// TwinCAT 3 PLC project RecipeServer_v2
// ProgramVersion: 3.1.4023.0
// libraries:
//   StringUtils, * (System)
//   Tc2_Standard, * (Beckhoff Automation GmbH)
//   Tc2_System, * (Beckhoff Automation GmbH)
//   Tc2_Utilities, * (Beckhoff Automation GmbH)
//   Tc3_Database, * (Beckhoff Automation GmbH)
//   Tc3_EventLogger, * (Beckhoff Automation GmbH)
//   Tc3_Module, * (Beckhoff Automation GmbH)
// project tree:
//   DUTs/Enumerations/ AllMaterialsEnum.TcTLEO
//   DUTs/ PaperInterval.TcDUT, PositionMaterials.TcDUT, PositionRotations.TcDUT, STRING_5K.TcDUT
//   GVLs/ BundleData.TcGVL, ExtrusionData.TcGVL, StrapWrapRecipe.TcGVL
//   GVLs/Constants/ GVL.TcGVL
//   / PlcTask.TcTTO
//   POUs/ AddRecipeToDatabase.TcPOU, MAIN.TcPOU, Validation.TcPOU
//   POUs/Functions/ ArrayFunctions.TcPOU, ConcatStrings.TcPOU
// (motion and I/O tree: see PLC project newplc)
// real-time tasks:
//   TASK PlcTask: cycle T#10ms, priority 20, ADS port 350
//   TASK PlcTask1: cycle T#10ms, priority 21, ADS port 351
//   TASK PlcTask2: cycle T#10ms, priority 22, ADS port 352
//   TASK PlcTask3: cycle T#10ms, priority 23, ADS port 353
//   TASK PlcTask4: cycle T#10ms, priority 24, ADS port 354
//   TASK PlcTask5: cycle T#10ms, priority 25, ADS port 355

CONFIGURATION RecipeServer_v2
    RESOURCE PLC ON TwinCAT3
        TASK PlcTask(INTERVAL := T#10ms, PRIORITY := 25);
        PROGRAM MAIN WITH PlcTask : MAIN;
    END_RESOURCE
END_CONFIGURATION

// ---- DUTs/Enumerations/AllMaterialsEnum.TcTLEO
{attribute 'qualified_only'}
{attribute 'strict'}
{attribute 'to_string'}
TYPE AllMaterialsEnum :
(
	//SIDES
	TOP, SIDES, BOTTOM,

	//CARDBOARD
	CAR20S, CAR20M, CAR20L, CAR28S, CAR28M, CAR28L, //base (flat)
	CAR20SF, CAR20MF, CAR20LF, CAR28SF, CAR28MF, CAR28LF, //single folded (L shape) - F
	CAR20SD, CAR20MD, CAR20LD, CAR28SD, CAR28MD, CAR28LD, //double folded (C shape) - D
	
	//CHIPBOARD
	CIP18, CIP54,
	
	//CORNER GUARD
	COR48,
	
	//PAPER
	PAP28,
	
	//WOOD BUNK
	WDT20, WDT22, WDT28, //top
	WDB20, WDB22, WDB28, //bottom
	WDS08, WDS10, WDS12, WDS14, WDS20, WDS22, WDS28, //side
	WDS8X8, WDS8X10, WDS12X12, WDS12X14, WDS20X10, WDS20X12, //side combined - X
	WDW20, WDW22, //special top (wide)
	
	size //number of materials
);
END_TYPE

// ---- DUTs/PaperInterval.TcDUT
TYPE PaperInterval :
STRUCT
	start : INT;
	end : INT;
	
	wrap : BOOL;
END_STRUCT
END_TYPE

// ---- DUTs/PositionMaterials.TcDUT
TYPE PositionMaterials :
STRUCT
	position : INT := 0; //default value is set to predefined constant if bundle needs less than 32 position material pairs
	
	top : STRING;
	left : STRING;
	right : STRING;
	bottom : STRING;
	
	topLeft : STRING;
	topLeftFold : INT;
	
	topRight : STRING;
	topRightFold : INT;
	
	bottomLeft : STRING;
	bottomLeftFold : INT;
	
	bottomRight : STRING;
	bottomRightFold : INT;
	
	numWrapPoints : INT;
	numWrapRotations : INT;
	
END_STRUCT
END_TYPE

// ---- DUTs/PositionRotations.TcDUT
TYPE PositionRotations : 
STRUCT
	position : INT;
	rotations : INT;
END_STRUCT
END_TYPE

// ---- DUTs/STRING_5K.TcDUT
TYPE STRING_5K : STRING(5000); END_TYPE

// ---- GVLs/BundleData.TcGVL
{attribute 'qualified_only'}
VAR_GLOBAL
	id : STRING;
	weight : REAL;
	
	length : REAL;
	height : REAL;
	width : REAL;
	
	pieces : USINT;
	layers : USINT;
	piecesPerLayer : USINT;
	
	requiredProcessing : ARRAY[0..3] OF BOOL;
END_VAR
VAR_GLOBAL CONSTANT
	//for requiredProcessing array
	AUTO_RE : INT := 0;
	MANUAL_RE : INT := 1;
	AUTO_SS : INT := 2;
	MANUAL_SS : INT := 3;
END_VAR

// ---- GVLs/ExtrusionData.TcGVL
{attribute 'qualified_only'}
VAR_GLOBAL	
	extrusionWeight : REAL;
	
	extrusionHeight : REAL;
	extrusionWidth : REAL;
END_VAR

// ---- GVLs/Constants/GVL.TcGVL
{attribute 'qualified_only'}
{attribute 'global_init_slot' := '45000'}
VAR_GLOBAL CONSTANT //first to compile
	maxMessages : UINT := 64;
	maxMaterials : DINT := 16; //max index, 0-15 are used with 16 as buffer
	
	//by materials
	Paper : ARRAY[1..1] OF STRING := ['PAP28'];
	CornerGuard : ARRAY[1..2] OF STRING := ['COR48', 'COR96'];
	
	CardboardSurfaces : ARRAY[1..6] OF STRING := ['CAR20S', 'CAR20M', 'CAR20L', 'CAR28S', 'CAR28M', 'CAR28L'];
	CardboardCorners : ARRAY[1..6] OF STRING := ['CAR20SF', 'CAR20MF', 'CAR20LF', 'CAR28SF', 'CAR28MF', 'CAR28LF'];
	
	Chipboard : ARRAY[1..2] OF STRING := ['CIP18', 'CIP54'];
	
	WoodBunkTop : ARRAY[1..5] OF STRING := ['WDT20', 'WDT22', 'WDT28', 'WDW20', 'WDW22'];
	WoodBunkSides : ARRAY[1..13] OF STRING := [	'WDS08', 'WDS10', 'WDS12', 'WDS14', 'WDS20','WDS22', 'WDS28', 'WDS8x8', 'WDS8x10', 'WDS12x12', 'WDS12x14', 'WDS20x10', 'WDS20x12'];										
	WoodBunkBottom : ARRAY[1..3] OF STRING := [	'WDB20', 'WDB22', 'WDB28'];
END_VAR

// ---- GVLs/StrapWrapRecipe.TcGVL
{attribute 'qualified_only'}
VAR_GLOBAL	
	//v2 - entries are in the format of position-material separated by material type
	faceCardboard : ARRAY[0..1] OF BOOL;
	facePaper : ARRAY[0..1] OF BOOL;
	
	TopPaper : ARRAY[0..GVL.maxMaterials] OF PaperInterval;
	LeftPaper : ARRAY[0..GVL.maxMaterials] OF PaperInterval;
	RightPaper : ARRAY[0..GVL.maxMaterials] OF PaperInterval;
	BottomPaper : ARRAY[0..GVL.maxMaterials] OF PaperInterval;
	
	Cardboard : ARRAY[0..GVL.maxMaterials] OF PositionMaterials;
	CornerGuard : ARRAY[0..GVL.maxMaterials] OF PositionMaterials;
	
	Chipboard : ARRAY[0..GVL.maxMaterials] OF PositionMaterials;
	WoodBunk : ARRAY[0..GVL.maxMaterials] OF PositionMaterials;
	
	PaperWrap : ARRAY[0..GVL.maxMaterials] OF PositionRotations;
	CardboardWrap : ARRAY[0..GVL.maxMaterials] OF PositionRotations;
END_VAR

// ---- POUs/MAIN.TcPOU
PROGRAM MAIN
VAR	
	generateRecipe : BOOL;
	
	addRecipeToDB : AddRecipeToDatabase;
	validator : Validation;
	arrayHelpers : ArrayFunctions;
	
	resetAddRecipeToDatabase : AddRecipeToDatabase;
	resetValidation : Validation;
	resetArrayFunctions : ArrayFunctions;
	
	start : BOOL := TRUE;
END_VAR

validator(); //real time error/warning message generator

IF generateRecipe THEN
	addRecipeToDB();
	
	IF addRecipeToDB.finished THEN
		reset();
		//reset all variables
		generateRecipe := FALSE;
		RETURN;
	END_IF
END_IF

METHOD reset : BOOL
VAR_INPUT
END_VAR
//reset FBs
MEMCPY(ADR(addRecipeToDB), ADR(resetAddRecipeToDatabase), SIZEOF(AddRecipeToDatabase));
MEMCPY(ADR(validator), ADR(resetValidation), SIZEOF(Validation));
MEMCPY(ADR(arrayHelpers), ADR(resetArrayFunctions), SIZEOF(ArrayFunctions));

//reset fields
BundleData.id := '';
BundleData.weight := 0;
BundleData.length := 0;
BundleData.height := 0;
BundleData.width := 0;
BundleData.pieces := 0;
BundleData.layers := 0;
BundleData.piecesPerLayer := 0;
MEMSET(ADR(BundleData.requiredProcessing), 0, SIZEOF(BundleData.requiredProcessing));

ExtrusionData.extrusionWeight := 0;
ExtrusionData.extrusionHeight := 0;
ExtrusionData.extrusionWidth := 0;

MEMSET(ADR(StrapWrapRecipe.facePaper), 0, SIZEOF(StrapWrapRecipe.facePaper));
MEMSET(ADR(StrapWrapRecipe.faceCardboard), 0, SIZEOF(StrapWrapRecipe.faceCardboard));
MEMSET(ADR(StrapWrapRecipe.TopPaper), 0, SIZEOF(StrapWrapRecipe.TopPaper));
MEMSET(ADR(StrapWrapRecipe.LeftPaper), 0, SIZEOF(StrapWrapRecipe.LeftPaper));
MEMSET(ADR(StrapWrapRecipe.RightPaper), 0, SIZEOF(StrapWrapRecipe.RightPaper));
MEMSET(ADR(StrapWrapRecipe.BottomPaper), 0, SIZEOF(StrapWrapRecipe.BottomPaper));
MEMSET(ADR(StrapWrapRecipe.Cardboard), 0, SIZEOF(StrapWrapRecipe.Cardboard));
MEMSET(ADR(StrapWrapRecipe.CornerGuard), 0, SIZEOF(StrapWrapRecipe.CornerGuard));
MEMSET(ADR(StrapWrapRecipe.Chipboard), 0, SIZEOF(StrapWrapRecipe.Chipboard));
MEMSET(ADR(StrapWrapRecipe.WoodBunk), 0, SIZEOF(StrapWrapRecipe.WoodBunk));
END_METHOD

END_PROGRAM

// ---- POUs/AddRecipeToDatabase.TcPOU
FUNCTION_BLOCK AddRecipeToDatabase //IMPLEMENTS I_TcEventBase
VAR
	cmd : ARRAY[0..19] OF STRING_5K;
	query : STRING_5K;
	
	fbSQLCommand : FB_SQLCommandEvt(sNetID := '', tTimeout := T#5S);
	fbSQLDatabase : FB_SQLDatabaseEvt (sNetID := '', tTimeout := T#5S);
	fbSQLResult: FB_SQLResultEvt(sNetID:='', tTimeout:=T#5S);
	
	eventString : STRING_5K;
	
	step : (CONNECT, READY, EXECUTE, FINISH);
END_VAR
VAR_OUTPUT
	finished : BOOL;
END_VAR

CASE step OF
	CONNECT:
		IF fbSQLDatabase.Connect(1) THEN
			IF NOT fbSqlDatabase.bError THEN
				step := READY;
			END_IF
		END_IF
		
	READY:
		IF fbSQLDatabase.CreateCmd(ADR(fbSQLCommand)) THEN
			step := EXECUTE;
		END_IF
	
	EXECUTE:
		query := completeQuery();
		IF fbSQLCommand.Execute(ADR(query), SIZEOF(query)) THEN
			step := FINISH;
		END_IF
		
	FINISH:
		IF fbSQLDatabase.Disconnect() THEN
			finished := TRUE;
		END_IF
END_CASE

METHOD completeQuery : STRING_5K
VAR_INST
	reqProcess : ARRAY[0..3] OF STRING_5K;
	
	queryOpening : STRING_5K := 'INSERT INTO "Bundle Data - Prototype" (BundleID, Weight, Length, Height, Width, Pieces, Layers, PiecesPerLayer, ExtrusionWeight, ExtrusionHeight, ExtrusionWidth, RequiredProcesses, Paper_top, Paper_sides, Paper_bottom, Cardboard, CornerGuard, Chipboard, WoodBunk) VALUES (';;
	queryClosing : STRING_5K := ')';
END_VAR
reqProcess[0] := TO_STRING(BundleData.requiredProcessing[0]);
reqProcess[1] := TO_STRING(BundleData.requiredProcessing[1]);
reqProcess[2] := TO_STRING(BundleData.requiredProcessing[2]);
reqProcess[3] := TO_STRING(BundleData.requiredProcessing[3]);


cmd[0] := TO_STRING(BundleData.id);
CONCAT2(ADR('$''), ADR(cmd[0]), ADR(cmd[0]), SIZEOF(cmd[0]));
CONCAT2(ADR(cmd[0]), ADR('$''), ADR(cmd[0]), SIZEOF(cmd[0]));

cmd[1] := TO_STRING(BundleData.weight);
cmd[2] := TO_STRING(BundleData.length);
cmd[3] := TO_STRING(BundleData.height);
cmd[4] := TO_STRING(BundleData.width);
cmd[5] := TO_STRING(BundleData.pieces);
cmd[6] := TO_STRING(BundleData.layers);
cmd[7] := TO_STRING(BundleData.piecesPerLayer);

cmd[8] := TO_STRING(ExtrusionData.extrusionWeight);
cmd[9] := TO_STRING(ExtrusionData.extrusionHeight);
cmd[10] := TO_STRING(ExtrusionData.extrusionWidth);

cmd[11] := ConcatStrings(reqProcess, 'ARRAY[', ']', ',');
//strap wrap recipe
cmd[12] := paperQuery(StrapWrapRecipe.TopPaper); //Paper_top
cmd[13] := paperQuery(StrapWrapRecipe.LeftPaper); //Paper_sides
cmd[14] := paperQuery(StrapWrapRecipe.RightPaper); //Paper_sides
cmd[15] := paperQuery(StrapWrapRecipe.BottomPaper); //Paper_sides

cmd[16] := materialQuery(StrapWrapRecipe.Cardboard);
cmd[17] := materialQuery(StrapWrapRecipe.CornerGuard);
cmd[18] := materialQuery(StrapWrapRecipe.Chipboard);
cmd[19] := materialQuery(StrapWrapRecipe.WoodBunk);

completeQuery := ConcatStrings(cmd, queryOpening, queryClosing, ',');
END_METHOD

METHOD materialQuery : STRING_5K
VAR_IN_OUT
	materialArr : ARRAY[*] OF PositionMaterials;
END_VAR
VAR_INST
	tempQuery : STRING_5K;
	
	position : STRING;
	top : STRING;
	left : STRING;
	right : STRING;
	bottom : STRING;
	
	topLeft : STRING;
	topLeftFold : STRING;
	topRight : STRING;
	topRightFold : STRING;
	
	bottomLeft : STRING;
	bottomLeftFold : STRING;
	bottomRight : STRING;
	bottomRightFold : STRING;
	
	i : DINT;
END_VAR
tempQuery := 'ARRAY[';

FOR i:=LOWER_BOUND(materialArr, 1) TO UPPER_BOUND(materialArr, 1) BY 1 DO
	position := TO_STRING(materialArr[i].position);
	
	top := TO_STRING(materialArr[i].top);
	left := TO_STRING(materialArr[i].left);
	right := TO_STRING(materialArr[i].right);
	bottom := TO_STRING(materialArr[i].bottom);
	
	topLeft := TO_STRING(materialArr[i].topLeft);
	topRight := TO_STRING(materialArr[i].topRight);
	bottomLeft := TO_STRING(materialArr[i].bottomLeft);
	bottomRight := TO_STRING(materialArr[i].bottomRight);
	
	topLeftFold := TO_STRING(materialArr[i].topLeftFold);
	topRightFold := TO_STRING(materialArr[i].topRightFold);
	bottomLeftFold := TO_STRING(materialArr[i].bottomLeftFold);
	bottomRightFold := TO_STRING(materialArr[i].bottomRightFold);
	
	IF top = '' AND left = '' AND right = '' AND bottom = '' AND topLeft = '' AND topRight = '' AND bottomLeft = '' AND bottomRight = '' THEN
		CONTINUE;
	END_IF
	
	IF i > LOWER_BOUND(materialArr, 1) THEN
		CONCAT2(ADR(tempQuery), ADR(', '), ADR(tempQuery), SIZEOF(tempQuery));
	END_IF

	CONCAT2(ADR(tempQuery), ADR('('), ADR(tempQuery), SIZEOF(tempQuery));
	CONCAT2(ADR(tempQuery), ADR(position), ADR(tempQuery), SIZEOF(tempQuery));
	CONCAT2(ADR(tempQuery), ADR(',$''), ADR(tempQuery), SIZEOF(tempQuery));
	
	CONCAT2(ADR(tempQuery), ADR(top), ADR(tempQuery), SIZEOF(tempQuery));
	CONCAT2(ADR(tempQuery), ADR('$', $''), ADR(tempQuery), SIZEOF(tempQuery));
	CONCAT2(ADR(tempQuery), ADR(left), ADR(tempQuery), SIZEOF(tempQuery));
	CONCAT2(ADR(tempQuery), ADR('$', $''), ADR(tempQuery), SIZEOF(tempQuery));
	CONCAT2(ADR(tempQuery), ADR(right), ADR(tempQuery), SIZEOF(tempQuery));
	CONCAT2(ADR(tempQuery), ADR('$', $''), ADR(tempQuery), SIZEOF(tempQuery));
	CONCAT2(ADR(tempQuery), ADR(bottom), ADR(tempQuery), SIZEOF(tempQuery));
	CONCAT2(ADR(tempQuery), ADR('$', $''), ADR(tempQuery), SIZEOF(tempQuery));
	
	CONCAT2(ADR(tempQuery), ADR(topLeft), ADR(tempQuery), SIZEOF(tempQuery));
	CONCAT2(ADR(tempQuery), ADR('$', $''), ADR(tempQuery), SIZEOF(tempQuery));
	CONCAT2(ADR(tempQuery), ADR(topRight), ADR(tempQuery), SIZEOF(tempQuery));
	CONCAT2(ADR(tempQuery), ADR('$', $''), ADR(tempQuery), SIZEOF(tempQuery));
	CONCAT2(ADR(tempQuery), ADR(bottomLeft), ADR(tempQuery), SIZEOF(tempQuery));
	CONCAT2(ADR(tempQuery), ADR('$', $''), ADR(tempQuery), SIZEOF(tempQuery));
	CONCAT2(ADR(tempQuery), ADR(bottomRight), ADR(tempQuery), SIZEOF(tempQuery));
	CONCAT2(ADR(tempQuery), ADR('$', '), ADR(tempQuery), SIZEOF(tempQuery));
	
	CONCAT2(ADR(tempQuery), ADR(topLeftFold), ADR(tempQuery), SIZEOF(tempQuery));
	CONCAT2(ADR(tempQuery), ADR(', '), ADR(tempQuery), SIZEOF(tempQuery));
	CONCAT2(ADR(tempQuery), ADR(topRightFold), ADR(tempQuery), SIZEOF(tempQuery));
	CONCAT2(ADR(tempQuery), ADR(', '), ADR(tempQuery), SIZEOF(tempQuery));
	CONCAT2(ADR(tempQuery), ADR(bottomLeftFold), ADR(tempQuery), SIZEOF(tempQuery));
	CONCAT2(ADR(tempQuery), ADR(', '), ADR(tempQuery), SIZEOF(tempQuery));
	CONCAT2(ADR(tempQuery), ADR(bottomRightFold), ADR(tempQuery), SIZEOF(tempQuery));
	
	CONCAT2(ADR(tempQuery), ADR(')'), ADR(tempQuery), SIZEOF(tempQuery));
END_FOR
CONCAT2(ADR(tempQuery), ADR(']::"PositionMaterials"[]'), ADR(tempQuery), SIZEOF(tempQuery));

materialQuery := tempQuery;
END_METHOD

METHOD paperQuery : STRING_5K
VAR_IN_OUT
	paperArr : ARRAY[*] OF PaperInterval;
END_VAR
VAR_INST
	tempQuery : STRING_5K;
	i : DINT;
	start : STRING;
	end : STRING;
	wrap : STRING;
END_VAR
tempQuery := 'ARRAY[';

FOR i:=LOWER_BOUND(paperArr, 1) TO UPPER_BOUND(paperArr, 1) BY 1 DO
	start := TO_STRING(paperArr[i].start);
	end := TO_STRING(paperArr[i].end);
	wrap := TO_STRING(paperArr[i].wrap);
	
	IF start = '0' AND end = '0' AND wrap = 'FALSE' THEN
		CONTINUE;
	END_IF
	
	IF i > LOWER_BOUND(paperArr, 1) THEN
		CONCAT2(ADR(tempQuery), ADR(','), ADR(tempQuery), SIZEOF(tempQuery));
	END_IF

	CONCAT2(ADR(tempQuery), ADR('('), ADR(tempQuery), SIZEOF(tempQuery));
	CONCAT2(ADR(tempQuery), ADR(start), ADR(tempQuery), SIZEOF(tempQuery));
	CONCAT2(ADR(tempQuery), ADR(','), ADR(tempQuery), SIZEOF(tempQuery));
	CONCAT2(ADR(tempQuery), ADR(end), ADR(tempQuery), SIZEOF(tempQuery));
	CONCAT2(ADR(tempQuery), ADR(','), ADR(tempQuery), SIZEOF(tempQuery));
	CONCAT2(ADR(tempQuery), ADR(wrap), ADR(tempQuery), SIZEOF(tempQuery));
	CONCAT2(ADR(tempQuery), ADR(')'), ADR(tempQuery), SIZEOF(tempQuery));
END_FOR
CONCAT2(ADR(tempQuery), ADR(']::"PaperInterval"[]'), ADR(tempQuery), SIZEOF(tempQuery));

paperQuery := tempQuery;
END_METHOD

END_FUNCTION_BLOCK

// ---- POUs/Functions/ConcatStrings.TcPOU
FUNCTION ConcatStrings : STRING_5K
VAR_IN_OUT
	stringsArr : ARRAY[*] OF STRING_5K;
END_VAR
VAR_INPUT
	opening : STRING_5K;
	closing : STRING_5K;
	separator : STRING_5K;
END_VAR
VAR
	fullString : STRING_5K;
	i : DINT := 0;	
END_VAR

fullString := opening; //opening segment

FOR i:=LOWER_BOUND(stringsArr, 1) TO UPPER_BOUND(stringsArr, 1)-1 BY 1 DO //first element to 2nd last element
	CONCAT2(ADR(fullString), ADR(stringsArr[i]), ADR(fullString), SIZEOF(fullString));
	CONCAT2(ADR(fullString), ADR(separator), ADR(fullString), SIZEOF(fullString));
END_FOR
CONCAT2(ADR(fullString), ADR(stringsArr[UPPER_BOUND(stringsArr, 1)]), ADR(fullString), SIZEOF(fullString)); //final element

CONCAT2(ADR(fullString), ADR(closing), ADR(fullString), SIZEOF(fullString)); //closing segment

concatStrings := fullString;

END_FUNCTION

// ---- POUs/Validation.TcPOU
FUNCTION_BLOCK Validation
VAR
	errors : ARRAY[0..GVL.maxMessages] OF STRING_5K;
	warnings : ARRAY[0..GVL.maxMessages] OF STRING_5K;

	tempErrors : ARRAY[0..GVL.maxMessages] OF STRING_5K;
	tempWarnings : ARRAY[0..GVL.maxMessages] OF STRING_5K;
	numErr : INT;
	numWarn : INT;
	
	bundleExists : BOOL;
		
	dbCheckStep : (CONNECT, READY, EXECUTE, FINISH);
	validationStep : (CHECK_EXISTING_BUNDLE, VALIDATE_DATA, FINISH_VALIDATION);
END_VAR

CASE validationStep OF
	CHECK_EXISTING_BUNDLE:
		IF checkExistingBundles() THEN
			validationStep := VALIDATE_DATA;
		END_IF
	
	VALIDATE_DATA:
		validateGeneralData(); //general data
		validateProcess(); //required processing
		validateMaterials(); //recipe
		
		validationStep := FINISH_VALIDATION;
		
	FINISH_VALIDATION: //copy temp to ADS and clear temp
		MEMCPY(ADR(errors), ADR(tempErrors), SIZEOF(errors));
		MEMCPY(ADR(warnings), ADR(tempWarnings), SIZEOF(warnings));
		
		MEMSET(ADR(tempErrors), 0, SIZEOF(tempErrors));
		MEMSET(ADR(tempWarnings), 0, SIZEOF(tempWarnings));
		numErr := 0;
		numWarn := 0;
		
		validationStep := CHECK_EXISTING_BUNDLE;
END_CASE

METHOD checkExistingBundles : BOOL
VAR_INST
	fbSQLCommand : FB_SQLCommandEvt(sNetID := '', tTimeout := T#5S);
	fbSQLDatabase : FB_SQLDatabaseEvt(sNetID := '', tTimeout := T#5S);
	fbSQLResult: FB_SQLResultEvt(sNetID := '', tTimeout := T#5S);
	
	
	cmd : ARRAY[0..2] OF STRING_5K;
	query : STRING_5K;
	tcMessage : I_TcMessage;
	existingID : STRING;
END_VAR
CASE dbCheckStep OF
	CONNECT:
		IF fbSQLDatabase.Connect(1) THEN
			IF NOT fbSqlDatabase.bError THEN
				dbCheckStep := READY;
			END_IF
		END_IF
		
	READY:
		IF fbSQLDatabase.CreateCmd(ADR(fbSQLCommand)) THEN
			dbCheckStep := EXECUTE;
		END_IF
	
	EXECUTE:
		cmd[0] := 'SELECT BundleID FROM "Bundle Data - Prototype" WHERE BundleID = $'';
		cmd[1] := TO_STRING(BundleData.id);
		cmd[2] := '$'';
		query := ConcatStrings(cmd, '', '', '');
		
		IF fbSQLCommand.ExecuteDataReturn(ADR(query), SIZEOF(query), ADR(fbSqlResult)) THEN
			dbCheckStep := FINISH;
		END_IF
		
	FINISH:
		fbSqlResult.Read(0, 1, ADR(existingID), SIZEOF(existingID), TRUE, FALSE);
		IF BundleData.id = existingID THEN
			bundleExists := TRUE;
		ELSE
			bundleExists := FALSE;
		END_IF
		IF fbSQLDatabase.Disconnect() THEN
			fbSqlResult.Release();
			checkExistingBundles := TRUE;
			dbCheckStep := CONNECT;
		END_IF
END_CASE
END_METHOD

{attribute 'TcRpcEnable'}
METHOD validateCardboard : BOOL
VAR_INST
	i : DINT;
END_VAR
FOR i:=0 TO GVL.maxMaterials BY 1 DO
	IF i > 0 THEN
		IF
			StrapWrapRecipe.Cardboard[i].position = StrapWrapRecipe.Cardboard[i-1].position 
			AND
			NOT(StrapWrapRecipe.Cardboard[i].position = 0 OR StrapWrapRecipe.Cardboard[i-1].position = 0)
		THEN
			tempWarnings[numWarn] := 'Cardboard: duplicate position';
			numWarn := numWarn + 1;
		END_IF
	END_IF
END_FOR
END_METHOD

{attribute 'TcRpcEnable'}
METHOD validateChipboard : BOOL
VAR_INST
	i : DINT;
END_VAR
FOR i:=0 TO GVL.maxMaterials BY 1 DO
	IF i > 0 THEN
		IF 
			StrapWrapRecipe.Chipboard[i].position = StrapWrapRecipe.Chipboard[i-1].position 
			AND
			NOT(StrapWrapRecipe.Chipboard[i].position = 0 OR StrapWrapRecipe.Chipboard[i-1].position = 0)
		THEN
			tempWarnings[numWarn] := 'Chipboard: duplicate position';
			numWarn := numWarn + 1;
		END_IF
	END_IF
END_FOR
END_METHOD

{attribute 'TcRpcEnable'}
METHOD validateCornerGuard : BOOL
VAR_INST
	i : DINT;
END_VAR
FOR i:=0 TO GVL.maxMaterials BY 1 DO
	IF i > 0 THEN
		IF 
			StrapWrapRecipe.CornerGuard[i].position = StrapWrapRecipe.CornerGuard[i-1].position 
			AND
			NOT(StrapWrapRecipe.CornerGuard[i].position = 0 OR StrapWrapRecipe.CornerGuard[i-1].position = 0)
		THEN
			tempWarnings[numWarn] := 'Corner Guard: duplicate position';
			numWarn := numWarn + 1;
		END_IF
	END_IF
END_FOR
END_METHOD

METHOD validateGeneralData : BOOL
IF BundleData.id = '' THEN //bundle id
	tempErrors[numErr] := 'ID missing';
	numErr := numErr + 1;
ELSIF BundleData.id <> '' AND bundleExists THEN
	tempWarnings[numWarn] := 'Bundle with entered ID already exists, proceeding will overwrite the existing recipe';
	numWarn := numWarn + 1;
END_IF

IF BundleData.weight = 0 THEN
	tempErrors[numErr] := 'Bundle weight missing';
	numErr := numErr + 1;
END_IF
IF BundleData.length = 0 OR BundleData.height = 0 OR BundleData.width = 0 THEN
	tempErrors[numErr] := 'Bundle dimension(s) missing';
	numErr := numErr + 1;
END_IF
IF BundleData.pieces = 0 OR BundleData.layers = 0 OR BundleData.piecesPerLayer = 0 THEN
	tempErrors[numErr] := 'Bundle layer dimension(s) missing';
	numErr := numErr + 1;
END_IF

IF Extrusiondata.extrusionWeight = 0 THEN
	tempErrors[numErr] := 'Extrusion weight missing';
	numErr := numErr + 1;
END_IF

IF Extrusiondata.extrusionHeight = 0 OR Extrusiondata.extrusionWidth = 0 THEN
	tempErrors[numErr] := 'Extrusion dimension(s) missing';
	numErr := numErr + 1;
END_IF
END_METHOD

{attribute 'TcRpcEnable'}
METHOD validateMaterials : BOOL
VAR_INST
	//fbSQLCommand : FB_SQLCommandEvt(sNetID := '', tTimeout := T#5S);
	//fbSQLDatabase : FB_SQLDatabaseEvt (sNetID := '', tTimeout := T#5S);
	//fbSQLResult: FB_SQLResultEvt(sNetID:='', tTimeout:=T#5S);
	
	
	
	
	//sqlResult : FB_SQLResult;
	
END_VAR

validatePaper();
validateCardboard();
validateCornerGuard();
validateChipboard();
validateWoodBunk();
END_METHOD

{attribute 'TcRpcEnable'}
METHOD validatePaper : BOOL
VAR_INST
	i : DINT;
END_VAR
FOR i:=0 TO GVL.maxMaterials BY 1 DO
	IF StrapWrapRecipe.TopPaper[i].start = 0 AND StrapWrapRecipe.TopPaper[i].end = 0 THEN //unused entry, do nothing and skip
		CONTINUE;
	END_IF
	
	IF StrapWrapRecipe.TopPaper[i].start >= StrapWrapRecipe.TopPaper[i].end THEN //invalid interval where start > end
		tempErrors[numErr] := 'Paper (Top): Start position must be less than end position';
		numErr := numErr + 1;
	END_IF
	
	IF i > 0 THEN
		IF StrapWrapRecipe.TopPaper[i].start < StrapWrapRecipe.TopPaper[i-1].end AND StrapWrapRecipe.TopPaper[i-1].end > 0 THEN //overlaps
			tempWarnings[numWarn] := 'Paper (Top): Overlapping segments';
			numWarn := numWarn + 1;
		ELSIF StrapWrapRecipe.TopPaper[i].start = StrapWrapRecipe.TopPaper[i-1].end AND StrapWrapRecipe.TopPaper[i-1].end > 0 THEN //adjacency
			tempWarnings[numWarn] := 'Paper (Top): Adjacent segments';
			numWarn := numWarn + 1;
		END_IF
	END_IF
END_FOR

FOR i:=0 TO GVL.maxMaterials BY 1 DO
	IF StrapWrapRecipe.LeftPaper[i].start = 0 AND StrapWrapRecipe.LeftPaper[i].end = 0 THEN //unused entry, do nothing and skip
		CONTINUE;
	END_IF
	
	IF StrapWrapRecipe.LeftPaper[i].start >= StrapWrapRecipe.LeftPaper[i].end THEN //invalid interval where start > end
		tempErrors[numErr] := 'Paper (Left): Start position must be less than end position';
		numErr := numErr + 1;
	END_IF
	
	IF i > 0 THEN
		IF StrapWrapRecipe.LeftPaper[i].start < StrapWrapRecipe.LeftPaper[i-1].end AND StrapWrapRecipe.LeftPaper[i-1].end > 0 THEN //overlaps
			tempWarnings[numWarn] := 'Paper (Left): Overlapping intervals, ignore if this is intended';
			numWarn := numWarn + 1;
		ELSIF StrapWrapRecipe.LeftPaper[i].start = StrapWrapRecipe.LeftPaper[i-1].end AND StrapWrapRecipe.LeftPaper[i-1].end > 0 THEN //adjacency
			tempWarnings[numWarn] := 'Paper (Left): Adjacent intervals can connected, ignore if this is intended';
			numWarn := numWarn + 1;
		END_IF
	END_IF
END_FOR

FOR i:=0 TO GVL.maxMaterials BY 1 DO
	IF StrapWrapRecipe.RightPaper[i].start = 0 AND StrapWrapRecipe.RightPaper[i].end = 0 THEN //unused entry, do nothing and skip
		CONTINUE;
	END_IF
	
	IF StrapWrapRecipe.RightPaper[i].start >= StrapWrapRecipe.RightPaper[i].end THEN //invalid interval where start > end
		tempErrors[numErr] := 'Paper (Right): Start position must be less than end position';
		numErr := numErr + 1;
	END_IF
	
	IF i > 0 THEN
		IF StrapWrapRecipe.RightPaper[i].start < StrapWrapRecipe.RightPaper[i-1].end AND StrapWrapRecipe.RightPaper[i-1].end > 0 THEN //overlaps
			tempWarnings[numWarn] := 'Paper (Right): Overlapping intervals, ignore if this is intended';
			numWarn := numWarn + 1;
		ELSIF StrapWrapRecipe.RightPaper[i].start = StrapWrapRecipe.RightPaper[i-1].end AND StrapWrapRecipe.RightPaper[i-1].end > 0 THEN //adjacency
			tempWarnings[numWarn] := 'Paper (Right): Adjacent intervals can connected, ignore if this is intended';
			numWarn := numWarn + 1;
		END_IF
	END_IF
END_FOR

FOR i:=0 TO GVL.maxMaterials BY 1 DO
	IF StrapWrapRecipe.BottomPaper[i].start = 0 AND StrapWrapRecipe.BottomPaper[i].end = 0 THEN //unused entry, do nothing and skip
		CONTINUE;
	END_IF
	
	IF StrapWrapRecipe.BottomPaper[i].start >= StrapWrapRecipe.BottomPaper[i].end THEN //invalid interval where start > end
		tempErrors[numErr] := 'Paper (Bottom): Start position must be less than end position';
		numErr := numErr + 1;
	END_IF
	
	IF i > 0 THEN
		IF StrapWrapRecipe.BottomPaper[i].start < StrapWrapRecipe.BottomPaper[i-1].end AND StrapWrapRecipe.BottomPaper[i-1].end > 0 THEN //overlaps
			tempWarnings[numWarn] := 'Paper (Bottom): Overlapping segments';
			numWarn := numWarn + 1;
		ELSIF StrapWrapRecipe.BottomPaper[i].start = StrapWrapRecipe.BottomPaper[i-1].end AND StrapWrapRecipe.BottomPaper[i-1].end > 0 THEN //adjacency
			tempWarnings[numWarn] := 'Paper (Bottom): Adjacent segments';
			numWarn := numWarn + 1;
		END_IF
	END_IF
END_FOR
END_METHOD

METHOD validateProcess : BOOL
VAR_INPUT
END_VAR
IF ( //if recipe exists but auto/manual strap and wrap is not selected
	StrapWrapRecipe.TopPaper[0].end > 0 OR 
	StrapWrapRecipe.LeftPaper[0].end > 0 OR 
	StrapWrapRecipe.RightPaper[0].end > 0 OR
	StrapWrapRecipe.BottomPaper[0].end > 0 OR 
	
	StrapWrapRecipe.Cardboard[0].top <> '' OR 
	StrapWrapRecipe.Cardboard[0].left <> '' OR 
	StrapWrapRecipe.Cardboard[0].right <> '' OR 
	StrapWrapRecipe.Cardboard[0].bottom <> '' OR 
	
	StrapWrapRecipe.Cardboard[0].topLeft <> '' OR 
	StrapWrapRecipe.Cardboard[0].topRight <> '' OR 
	StrapWrapRecipe.Cardboard[0].bottomLeft <> '' OR 
	StrapWrapRecipe.Cardboard[0].bottomRight <> '' OR 
	
	StrapWrapRecipe.CornerGuard[0].topLeft <> '' OR 
	StrapWrapRecipe.CornerGuard[0].topRight <> '' OR 
	StrapWrapRecipe.CornerGuard[0].bottomLeft <> '' OR 
	StrapWrapRecipe.CornerGuard[0].bottomRight <> '' OR 
	
	StrapWrapRecipe.Chipboard[0].top <> '' OR 
	StrapWrapRecipe.Chipboard[0].left <> '' OR 
	StrapWrapRecipe.Chipboard[0].right <> '' OR 
	StrapWrapRecipe.Chipboard[0].Bottom <> '' OR 

	StrapWrapRecipe.WoodBunk[0].top <> '' OR 
	StrapWrapRecipe.WoodBunk[0].left <> '' OR 
	StrapWrapRecipe.WoodBunk[0].right <> '' OR 
	StrapWrapRecipe.WoodBunk[0].Bottom <> '')
THEN
	IF NOT BundleData.requiredProcessing[BundleData.AUTO_SS] AND NOT BundleData.requiredProcessing[BundleData.MANUAL_SS] THEN
		tempErrors[numErr] := 'Recipe exists but strap and wrap processes are not selected (Auto/Manual Strap and Wrap)';
		numErr := numErr + 1;
	END_IF
ELSE //no recipe exists but auto/manual strap and wrap is selected
	IF BundleData.requiredProcessing[BundleData.AUTO_SS] OR BundleData.requiredProcessing[BundleData.MANUAL_SS] THEN
		tempWarnings[numWarn] := 'Strap and wrap processes are selected but there is no recipe, is this intended?';
		numWarn := numWarn + 1;
	END_IF
END_IF

	
IF //auto and manual strap/wrap are both selected
	(BundleData.requiredProcessing[BundleData.AUTO_RE] AND BundleData.requiredProcessing[BundleData.MANUAL_RE]) OR
	(BundleData.requiredProcessing[BundleData.AUTO_SS] AND BundleData.requiredProcessing[BundleData.MANUAL_SS])
THEN
	tempErrors[numErr] := 'Auto and Manual processes of the same type cannot be selected together';
	numErr := numErr + 1;
	
ELSIF //no processes selected
	NOT BundleData.requiredProcessing[BundleData.AUTO_RE] AND 
	NOT BundleData.requiredProcessing[BundleData.AUTO_SS] AND
	NOT BundleData.requiredProcessing[BundleData.MANUAL_RE] AND 
	NOT BundleData.requiredProcessing[BundleData.MANUAL_SS]
THEN
	tempWarnings[numWarn] := 'No processes are selected, is this intended?';
	numWarn := numWarn + 1;
END_IF
END_METHOD

{attribute 'TcRpcEnable'}
METHOD validateWoodBunk : BOOL
VAR_INST
	i : DINT;
END_VAR
FOR i:=0 TO GVL.maxMaterials BY 1 DO
	IF i > 0 THEN
		IF 
			StrapWrapRecipe.WoodBunk[i].position = StrapWrapRecipe.WoodBunk[i-1].position 
			AND
			NOT(StrapWrapRecipe.WoodBunk[i].position = 0 OR StrapWrapRecipe.WoodBunk[i-1].position = 0)
		THEN
			tempWarnings[numWarn] := 'Wood Bunk: duplicate position';
			numWarn := numWarn + 1;
		END_IF
	END_IF
END_FOR
END_METHOD

END_FUNCTION_BLOCK

// ---- POUs/Functions/ArrayFunctions.TcPOU
FUNCTION_BLOCK ArrayFunctions
VAR
	j : DINT;
END_VAR

{attribute 'TcRpcEnable'}
METHOD removeCardboard : BOOL
VAR_INPUT
	i : INT; //index to be removed
END_VAR
MEMMOVE(ADR(StrapWrapRecipe.Cardboard[i]), ADR(StrapWrapRecipe.Cardboard[i+1]), (GVL.maxMaterials-i)*SIZEOF(PositionMaterials));
StrapWrapRecipe.Cardboard[GVL.maxMaterials].position := 0;

StrapWrapRecipe.Cardboard[GVL.maxMaterials].top := '';
StrapWrapRecipe.Cardboard[GVL.maxMaterials].left := '';
StrapWrapRecipe.Cardboard[GVL.maxMaterials].right := '';
StrapWrapRecipe.Cardboard[GVL.maxMaterials].bottom := '';

StrapWrapRecipe.Cardboard[GVL.maxMaterials].topLeft := '';
StrapWrapRecipe.Cardboard[GVL.maxMaterials].topRight := '';
StrapWrapRecipe.Cardboard[GVL.maxMaterials].bottomLeft := '';
StrapWrapRecipe.Cardboard[GVL.maxMaterials].bottomRight := '';

StrapWrapRecipe.Cardboard[GVL.maxMaterials].topLeftFold := 0;
StrapWrapRecipe.Cardboard[GVL.maxMaterials].topRightFold := 0;
StrapWrapRecipe.Cardboard[GVL.maxMaterials].bottomLeftFold := 0;
StrapWrapRecipe.Cardboard[GVL.maxMaterials].bottomRightFold := 0;
END_METHOD

{attribute 'TcRpcEnable'}
METHOD removeChipboard : BOOL
VAR_INPUT
	i : INT; //index to be removed
END_VAR
MEMMOVE(ADR(StrapWrapRecipe.Chipboard[i]), ADR(StrapWrapRecipe.Chipboard[i+1]), (GVL.maxMaterials-i)*SIZEOF(PositionMaterials));
StrapWrapRecipe.Chipboard[GVL.maxMaterials].position := 0;

StrapWrapRecipe.Chipboard[GVL.maxMaterials].top := '';
StrapWrapRecipe.Chipboard[GVL.maxMaterials].left := '';
StrapWrapRecipe.Chipboard[GVL.maxMaterials].right := '';
StrapWrapRecipe.Chipboard[GVL.maxMaterials].bottom := '';

StrapWrapRecipe.Chipboard[GVL.maxMaterials].topLeft := '';
StrapWrapRecipe.Chipboard[GVL.maxMaterials].topRight := '';
StrapWrapRecipe.Chipboard[GVL.maxMaterials].bottomLeft := '';
StrapWrapRecipe.Chipboard[GVL.maxMaterials].bottomRight := '';

StrapWrapRecipe.Chipboard[GVL.maxMaterials].topLeftFold := 0;
StrapWrapRecipe.Chipboard[GVL.maxMaterials].topRightFold := 0;
StrapWrapRecipe.Chipboard[GVL.maxMaterials].bottomLeftFold := 0;
StrapWrapRecipe.Chipboard[GVL.maxMaterials].bottomRightFold := 0;
END_METHOD

{attribute 'TcRpcEnable'}
METHOD removeCornerGuard : BOOL
VAR_INPUT
	i : INT; //index to be removed
END_VAR
MEMMOVE(ADR(StrapWrapRecipe.CornerGuard[i]), ADR(StrapWrapRecipe.CornerGuard[i+1]), (GVL.maxMaterials-i)*SIZEOF(PositionMaterials));
StrapWrapRecipe.CornerGuard[GVL.maxMaterials].position := 0;

MEMSET(ADR(StrapWrapRecipe.CornerGuard[GVL.maxMaterials]), 0, SIZEOF(PositionMaterials));
END_METHOD

{attribute 'TcRpcEnable'}
METHOD removePaper: BOOL
VAR_INPUT
	face : STRING;
	i : DINT; //index to be removed
END_VAR
IF face = 'Top' THEN
	MEMMOVE(ADR(StrapWrapRecipe.TopPaper[i]), ADR(StrapWrapRecipe.TopPaper[i+1]), (GVL.maxMaterials-i)*SIZEOF(PaperInterval));
	StrapWrapRecipe.TopPaper[GVL.maxMaterials].start := 0;
	StrapWrapRecipe.TopPaper[GVL.maxMaterials].end := 0;
ELSIF face = 'Left' THEN
	MEMMOVE(ADR(StrapWrapRecipe.LeftPaper[i]), ADR(StrapWrapRecipe.LeftPaper[i+1]), (GVL.maxMaterials-i)*SIZEOF(PaperInterval));
	StrapWrapRecipe.LeftPaper[GVL.maxMaterials].start := 0;
	StrapWrapRecipe.LeftPaper[GVL.maxMaterials].end := 0;
ELSIF face = 'Right' THEN
	MEMMOVE(ADR(StrapWrapRecipe.RightPaper[i]), ADR(StrapWrapRecipe.RightPaper[i+1]), (GVL.maxMaterials-i)*SIZEOF(PaperInterval));
	StrapWrapRecipe.RightPaper[GVL.maxMaterials].start := 0;
	StrapWrapRecipe.RightPaper[GVL.maxMaterials].end := 0;
ELSIF face = 'Bottom' THEN
	MEMMOVE(ADR(StrapWrapRecipe.TopPaper[i]), ADR(StrapWrapRecipe.TopPaper[i+1]), (GVL.maxMaterials-i)*SIZEOF(PaperInterval));
	StrapWrapRecipe.BottomPaper[GVL.maxMaterials].start := 0;
	StrapWrapRecipe.BottomPaper[GVL.maxMaterials].end := 0;
END_IF
END_METHOD

{attribute 'TcRpcEnable'}
METHOD removeWoodBunk : BOOL
VAR_INPUT
	i : INT; //index to be removed
END_VAR
MEMMOVE(ADR(StrapWrapRecipe.WoodBunk[i]), ADR(StrapWrapRecipe.WoodBunk[i+1]), (GVL.maxMaterials-i)*SIZEOF(PositionMaterials));
StrapWrapRecipe.WoodBunk[GVL.maxMaterials].position := 0;

StrapWrapRecipe.WoodBunk[GVL.maxMaterials].top := '';
StrapWrapRecipe.WoodBunk[GVL.maxMaterials].left := '';
StrapWrapRecipe.WoodBunk[GVL.maxMaterials].right := '';
StrapWrapRecipe.WoodBunk[GVL.maxMaterials].bottom := '';

StrapWrapRecipe.WoodBunk[GVL.maxMaterials].topLeft := '';
StrapWrapRecipe.WoodBunk[GVL.maxMaterials].topRight := '';
StrapWrapRecipe.WoodBunk[GVL.maxMaterials].bottomLeft := '';
StrapWrapRecipe.WoodBunk[GVL.maxMaterials].bottomRight := '';

StrapWrapRecipe.WoodBunk[GVL.maxMaterials].topLeftFold := 0;
StrapWrapRecipe.WoodBunk[GVL.maxMaterials].topRightFold := 0;
StrapWrapRecipe.WoodBunk[GVL.maxMaterials].bottomLeftFold := 0;
StrapWrapRecipe.WoodBunk[GVL.maxMaterials].bottomRightFold := 0;
END_METHOD

{attribute 'TcRpcEnable'}
METHOD sortEntries : BOOL
sortPositionMaterials(StrapWrapRecipe.Cardboard);
sortPositionMaterials(StrapWrapRecipe.CornerGuard);
sortPositionMaterials(StrapWrapRecipe.Chipboard);
sortPositionMaterials(StrapWrapRecipe.WoodBunk);

sortPaperIntervals(StrapWrapRecipe.TopPaper);
sortPaperIntervals(StrapWrapRecipe.LeftPaper);
sortPaperIntervals(StrapWrapRecipe.RightPaper);
sortPaperIntervals(StrapWrapRecipe.BottomPaper);
END_METHOD

METHOD sortPaperIntervals : BOOL
VAR_IN_OUT
	arr : ARRAY[*] OF PaperInterval;
END_VAR
VAR_INST
	i : DINT;
	j : DINT;
	temp : PaperInterval;
END_VAR
FOR i:=LOWER_BOUND(arr, 1) TO UPPER_BOUND(arr, 1) BY 1 DO
	FOR j:=LOWER_BOUND(arr, 1) TO UPPER_BOUND(arr, 1)-i-1 BY 1 DO
		IF 
			(arr[j].start = 0 AND arr[j].end = 0) //unused entry
			OR 
			arr[j].start > arr[j+1].start AND //out of order and both entries are valid
			NOT(arr[j+1].start = 0 AND arr[j+1].end = 0)
		THEN //unused entry or out of order
			MEMCPY(ADR(temp), ADR(arr[j]), SIZEOF(PaperInterval));
			MEMCPY(ADR(arr[j]), ADR(arr[j+1]), SIZEOF(PaperInterval));
			MEMCPY(ADR(arr[j+1]), ADR(temp), SIZEOF(PaperInterval));
		END_IF
	END_FOR
END_FOR
END_METHOD

METHOD sortPositionMaterials : BOOL
VAR_IN_OUT
	arr : ARRAY[*] OF PositionMaterials;
END_VAR
VAR_INST
	i : DINT;
	j : DINT;
	temp : PositionMaterials;
END_VAR
FOR i:=LOWER_BOUND(arr, 1) TO UPPER_BOUND(arr, 1)-1 BY 1 DO
	FOR j:=LOWER_BOUND(arr, 1) TO UPPER_BOUND(arr, 1)-i-1 BY 1 DO
		IF //unused entry
			arr[j].top = '' AND arr[j].left = '' AND arr[j].right = '' AND arr[j].bottom = '' AND 
			arr[j].topRight = '' AND arr[j].topLeft = '' AND arr[j].bottomRight = '' AND arr[j].bottomLeft = ''
		THEN //unused entry
			arr[j].position := 0; //set position to 0
			MEMCPY(ADR(temp), ADR(arr[j]), SIZEOF(PositionMaterials));
			MEMCPY(ADR(arr[j]), ADR(arr[j+1]), SIZEOF(PositionMaterials));
			MEMCPY(ADR(arr[j+1]), ADR(temp), SIZEOF(PositionMaterials));
		ELSIF //out of order and both entries are valid
			arr[j].position > arr[j+1].position AND 
			NOT(
				arr[j+1].top = '' AND arr[j+1].left = '' AND arr[j+1].right = '' AND arr[j+1].bottom = '' AND 
				arr[j+1].topRight = '' AND arr[j+1].topLeft = '' AND arr[j+1].bottomRight = '' AND arr[j+1].bottomLeft = '')
		THEN
			MEMCPY(ADR(temp), ADR(arr[j]), SIZEOF(PositionMaterials));
			MEMCPY(ADR(arr[j]), ADR(arr[j+1]), SIZEOF(PositionMaterials));
			MEMCPY(ADR(arr[j+1]), ADR(temp), SIZEOF(PositionMaterials));
		END_IF
	END_FOR
END_FOR
END_METHOD

END_FUNCTION_BLOCK
